(* Schneider Machine Expert - Basic project Prototype 2, file version 2.7.0.0 *)
(* ProjectInformations: Name=Nuevo proyecto *)

HARDWARE
  Cpu 0: TM221M16R/G
  EthernetConfiguration: NetworkName=M221, IpAllocationMode=FixedAddress, IpAddress=0.0.0.0, SubnetMask=0.0.0.0
  SerialLineConfiguration: Baud=Baud19200, Parity=ParityEven, DataBits=DataBits8, StopBits=StopBits1, PhysicalMedium=PhysicalMediumRs485, TransmissionMode=TransmissionModeModbusRtu, SlaveId=1, Addressing=SlaveAddressing
  MastTask: UsePeriodScanMode=false, PeriodScan=100
  FastTask: Period=255
  CpuBehavior: StartingMode=StartAsPreviousState, AutoSaveRamOnEeprom=true, WatchdogPeriod=250

SYMBOLS  (address, symbol, comment, settings)
  %M0       START_BUTTON
  %M1       RESET_BUTTON
  %M2       STOP_BUTTON
  %M3       EMERGENCY_BUTTON
  %M4       AUTO_SWITCH
  %M5       TYPE_2
  %M6       TYPE_3
  %M7       ENTRY_SENSOR
  %M8       OBJECT_SENSOR_1
  %M9       EXIT_SENSOR
  %M10      PERSON
  %M11      OBJECT_SENSOR_2
  %M12      T1_SENSOR
  %M13      T2_SENSOR
  %M14      T3_SENSOR
  %M15      ENTRY_CONVEYOR
  %M16      GRAB_1
  %M17      MIDDLE_CONVEYOR
  %M18      GRAB_2
  %M19      EXIT_CONVEYOR
  %M20      CURVE_CONVEYOR
  %M21      SELECTOR_CONVEYOR
  %M22      T1_CONVEYOR
  %M23      T2_CONVEYOR
  %M24      T3_CONVEYOR
  %M25      BELT_1
  %M26      BELT_2
  %M27      BELT_3
  %M28      PALLET
  %M29      RED
  %M30      YELLOW
  %M31      GREEN
  %M32      ALARM
  %M33      ENTRY
  %M100     INITIALIZE
  %M101     INITIAL_POS_1
  %M102     INITIAL_POS_2
  %M200     FLAG_AUTO
  %S21      SB_INITGRAFCET  "En el estado 1, este bit provoca una inicialización GRAFCET. Los pasos activos se desactivan y los pasos iniciales se activan"
  %X1       STATE_1
  %X2       STATE_2
  %X3       STATE_3
  %X4       STATE_4
  %X5       STATE_5
  %X6       STATE_6
  %X7       STATE_7
  %X8       STATE_8
  %X9       STATE_9
  %X10      STATE_10
  %X11      STATE_11
  %X12      STATE_12
  %X13      STATE_13
  %X14      STATE_14
  %X15      STATE_15
  %X16      STATE_16
  %X17      STATE_17
  %X18      STATE_18
  %X19      STATE_19
  %X21      STATE_21
  %MW0      X1
  %MW1      Y1
  %MW2      Z1
  %MW3      X2
  %MW4      Y2
  %MW5      Z2
  %MW6      X1_MOVE
  %MW7      Y1_MOVE
  %MW8      Z1_MOVE
  %MW9      X2_MOVE
  %MW10     Y2_MOVE
  %MW11     Z2_MOVE
  %MW12     T1
  %MW13     T2
  %MW14     T3
  %TM0      TIME_TO_UNGRAB  [Preset=1, Base=OneHundredMilliSeconds]
  %TM1      SECURITY_TIME  [Preset=5, Base=OneSecond]
  %TM2      TIME_TO_WAIT_NEXT  [Preset=2, Base=OneSecond]
  %C0       T1_ITEMS
  %C1       T2_ITEMS
  %C2       T3_ITEMS

GRAFCET Grafcet
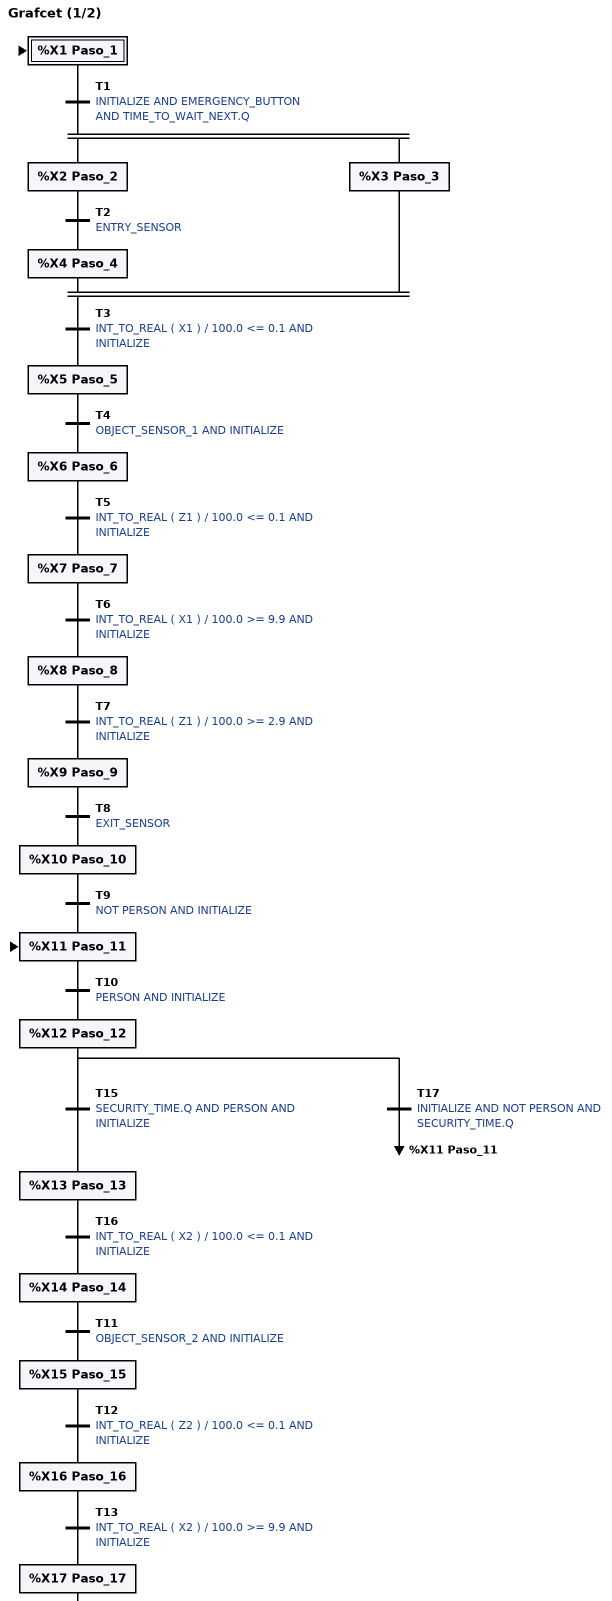
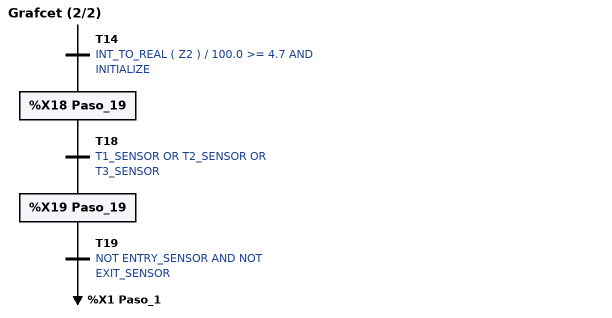
  INITIAL_STEP %X1  (* Paso_1 *)
  STEP %X2  (* Paso_2 *)
  STEP %X3  (* Paso_3 *)
  STEP %X4  (* Paso_4 *)
  STEP %X5  (* Paso_5 *)
  STEP %X6  (* Paso_6 *)
  STEP %X7  (* Paso_7 *)
  STEP %X8  (* Paso_8 *)
  STEP %X9  (* Paso_9 *)
  STEP %X10  (* Paso_10 *)
  STEP %X11  (* Paso_11 *)
  STEP %X12  (* Paso_12 *)
  STEP %X13  (* Paso_13 *)
  STEP %X14  (* Paso_14 *)
  STEP %X15  (* Paso_15 *)
  STEP %X16  (* Paso_16 *)
  STEP %X17  (* Paso_17 *)
  STEP %X18  (* Paso_19 *)
  STEP %X19  (* Paso_19 *)
  TRANSITION T1 FROM %X1 TO %X2, %X3 := INITIALIZE AND EMERGENCY_BUTTON AND TIME_TO_WAIT_NEXT.Q;
  TRANSITION T2 FROM %X2 TO %X4 := ENTRY_SENSOR;
  TRANSITION T3 FROM %X4, %X3 TO %X5 := INT_TO_REAL ( X1 ) / 100.0 <= 0.1 AND INITIALIZE;
  TRANSITION T4 FROM %X5 TO %X6 := OBJECT_SENSOR_1 AND INITIALIZE;
  TRANSITION T5 FROM %X6 TO %X7 := INT_TO_REAL ( Z1 ) / 100.0 <= 0.1 AND INITIALIZE;
  TRANSITION T6 FROM %X7 TO %X8 := INT_TO_REAL ( X1 ) / 100.0 >= 9.9 AND INITIALIZE;
  TRANSITION T7 FROM %X8 TO %X9 := INT_TO_REAL ( Z1 ) / 100.0 >= 2.9 AND INITIALIZE;
  TRANSITION T8 FROM %X9 TO %X10 := EXIT_SENSOR;
  TRANSITION T9 FROM %X10 TO %X11 := NOT PERSON AND INITIALIZE;
  TRANSITION T10 FROM %X11 TO %X12 := PERSON AND INITIALIZE;
  TRANSITION T11 FROM %X14 TO %X15 := OBJECT_SENSOR_2 AND INITIALIZE;
  TRANSITION T12 FROM %X15 TO %X16 := INT_TO_REAL ( Z2 ) / 100.0 <= 0.1 AND INITIALIZE;
  TRANSITION T13 FROM %X16 TO %X17 := INT_TO_REAL ( X2 ) / 100.0 >= 9.9 AND INITIALIZE;
  TRANSITION T14 FROM %X17 TO %X18 := INT_TO_REAL ( Z2 ) / 100.0 >= 4.7 AND INITIALIZE;
  TRANSITION T15 FROM %X12 TO %X13 := SECURITY_TIME.Q AND PERSON AND INITIALIZE;
  TRANSITION T16 FROM %X13 TO %X14 := INT_TO_REAL ( X2 ) / 100.0 <= 0.1 AND INITIALIZE;
  TRANSITION T17 FROM %X12 TO %X11 := INITIALIZE AND NOT PERSON AND SECURITY_TIME.Q;
  TRANSITION T18 FROM %X18 TO %X19 := T1_SENSOR OR T2_SENSOR OR T3_SENSOR;
  TRANSITION T19 FROM %X19 TO %X1 := NOT ENTRY_SENSOR AND NOT EXIT_SENSOR;

TRANSITION T1 (%X1 -> %X2, %X3) 
  (* SectionNumber=0 *)

// Rung 0: Tr1
  LD %M100                (* INITIALIZE *)
  AND %M3                 (* EMERGENCY_BUTTON *)
  AND %TM2.Q              (* TIME_TO_WAIT_NEXT *)
  ENDT
  // as ST:
  //   TRANSITION := INITIALIZE AND EMERGENCY_BUTTON AND TIME_TO_WAIT_NEXT.Q;

TRANSITION T2 (%X2 -> %X4) 
  (* SectionNumber=0 *)

// Rung 1: Tr2
  LD %M7                  (* ENTRY_SENSOR *)
  ENDT
  // as ST:
  //   TRANSITION := ENTRY_SENSOR;

TRANSITION T3 (%X4, %X3 -> %X5) 
  (* SectionNumber=0 *)

// Rung 2: Tr3
  LD 1
  AND [ INT_TO_REAL ( %MW0 ) / 100.0 <= 0.1 ](* X1 *)
  AND %M100               (* INITIALIZE *)
  ENDT
  // as ST:
  //   TRANSITION := INT_TO_REAL ( X1 ) / 100.0 <= 0.1 AND INITIALIZE;

TRANSITION T4 (%X5 -> %X6) 
  (* SectionNumber=0 *)

// Rung 3: Tr4
  LD %M8                  (* OBJECT_SENSOR_1 *)
  AND %M100               (* INITIALIZE *)
  ENDT
  // as ST:
  //   TRANSITION := OBJECT_SENSOR_1 AND INITIALIZE;

TRANSITION T5 (%X6 -> %X7) 
  (* SectionNumber=0 *)

// Rung 4: Tr5
  LD 1
  AND [ INT_TO_REAL ( %MW2 ) / 100.0 <= 0.1 ](* Z1 *)
  AND %M100               (* INITIALIZE *)
  ENDT
  // as ST:
  //   TRANSITION := INT_TO_REAL ( Z1 ) / 100.0 <= 0.1 AND INITIALIZE;

TRANSITION T6 (%X7 -> %X8) 
  (* SectionNumber=0 *)

// Rung 5: Tr6
  LD 1
  AND [ INT_TO_REAL ( %MW0 ) / 100.0 >= 9.9 ](* X1 *)
  AND %M100               (* INITIALIZE *)
  ENDT
  // as ST:
  //   TRANSITION := INT_TO_REAL ( X1 ) / 100.0 >= 9.9 AND INITIALIZE;

TRANSITION T7 (%X8 -> %X9) 
  (* SectionNumber=0 *)

// Rung 6: Tr7
  LD 1
  AND [ INT_TO_REAL ( %MW2 ) / 100.0 >= 2.9 ](* Z1 *)
  AND %M100               (* INITIALIZE *)
  ENDT
  // as ST:
  //   TRANSITION := INT_TO_REAL ( Z1 ) / 100.0 >= 2.9 AND INITIALIZE;

TRANSITION T8 (%X9 -> %X10) 
  (* SectionNumber=0 *)

// Rung 7: Tr8
  LD %M9                  (* EXIT_SENSOR *)
  ENDT
  // as ST:
  //   TRANSITION := EXIT_SENSOR;

TRANSITION T9 (%X10 -> %X11) 
  (* SectionNumber=0 *)

// Rung 8: Tr9
  LDN %M10                (* PERSON *)
  AND %M100               (* INITIALIZE *)
  ENDT
  // as ST:
  //   TRANSITION := NOT PERSON AND INITIALIZE;

TRANSITION T10 (%X11 -> %X12) 
  (* SectionNumber=0 *)

// Rung 9: Tr10
  LD %M10                 (* PERSON *)
  AND %M100               (* INITIALIZE *)
  ENDT
  // as ST:
  //   TRANSITION := PERSON AND INITIALIZE;

TRANSITION T11 (%X14 -> %X15) 
  (* SectionNumber=0 *)

// Rung 10: Tr14
  LD %M11                 (* OBJECT_SENSOR_2 *)
  AND %M100               (* INITIALIZE *)
  ENDT
  // as ST:
  //   TRANSITION := OBJECT_SENSOR_2 AND INITIALIZE;

TRANSITION T12 (%X15 -> %X16) 
  (* SectionNumber=0 *)

// Rung 11: Tr15
  LD 1
  AND [ INT_TO_REAL ( %MW5 ) / 100.0 <= 0.1 ](* Z2 *)
  AND %M100               (* INITIALIZE *)
  ENDT
  // as ST:
  //   TRANSITION := INT_TO_REAL ( Z2 ) / 100.0 <= 0.1 AND INITIALIZE;

TRANSITION T13 (%X16 -> %X17) 
  (* SectionNumber=0 *)

// Rung 12: Tr16
  LD 1
  AND [ INT_TO_REAL ( %MW3 ) / 100.0 >= 9.9 ](* X2 *)
  AND %M100               (* INITIALIZE *)
  ENDT
  // as ST:
  //   TRANSITION := INT_TO_REAL ( X2 ) / 100.0 >= 9.9 AND INITIALIZE;

TRANSITION T14 (%X17 -> %X18) 
  (* SectionNumber=0 *)

// Rung 13: Tr17
  LD 1
  AND [ INT_TO_REAL ( %MW5 ) / 100.0 >= 4.7 ](* Z2 *)
  AND %M100               (* INITIALIZE *)
  ENDT
  // as ST:
  //   TRANSITION := INT_TO_REAL ( Z2 ) / 100.0 >= 4.7 AND INITIALIZE;

TRANSITION T15 (%X12 -> %X13) 
  (* SectionNumber=0 *)

// Rung 14: Tr12
  LD %TM1.Q               (* SECURITY_TIME *)
  AND %M10                (* PERSON *)
  AND %M100               (* INITIALIZE *)
  ENDT
  // as ST:
  //   TRANSITION := SECURITY_TIME.Q AND PERSON AND INITIALIZE;

TRANSITION T16 (%X13 -> %X14) 
  (* SectionNumber=0 *)

// Rung 15: Tr13
  LD 1
  AND [ INT_TO_REAL ( %MW3 ) / 100.0 <= 0.1 ](* X2 *)
  AND %M100               (* INITIALIZE *)
  ENDT
  // as ST:
  //   TRANSITION := INT_TO_REAL ( X2 ) / 100.0 <= 0.1 AND INITIALIZE;

TRANSITION T17 (%X12 -> %X11) 
  (* SectionNumber=0 *)

// Rung 16: Tr11
  LD %M100                (* INITIALIZE *)
  ANDN %M10               (* PERSON *)
  AND %TM1.Q              (* SECURITY_TIME *)
  ENDT
  // as ST:
  //   TRANSITION := INITIALIZE AND NOT PERSON AND SECURITY_TIME.Q;

TRANSITION T18 (%X18 -> %X19) 
  (* SectionNumber=0 *)

// Rung 17: Tr18
  LD %M12                 (* T1_SENSOR *)
  OR %M13                 (* T2_SENSOR *)
  OR %M14                 (* T3_SENSOR *)
  ENDT
  // as ST:
  //   TRANSITION := T1_SENSOR OR T2_SENSOR OR T3_SENSOR;

TRANSITION T19 (%X19 -> %X1) 
  (* SectionNumber=0 *)

// Rung 18: Tr19
  LDN %M7                 (* ENTRY_SENSOR *)
  ANDN %M9                (* EXIT_SENSOR *)
  ENDT
  // as ST:
  //   TRANSITION := NOT ENTRY_SENSOR AND NOT EXIT_SENSOR;

POU Actions
  (* SectionNumber=21 *)

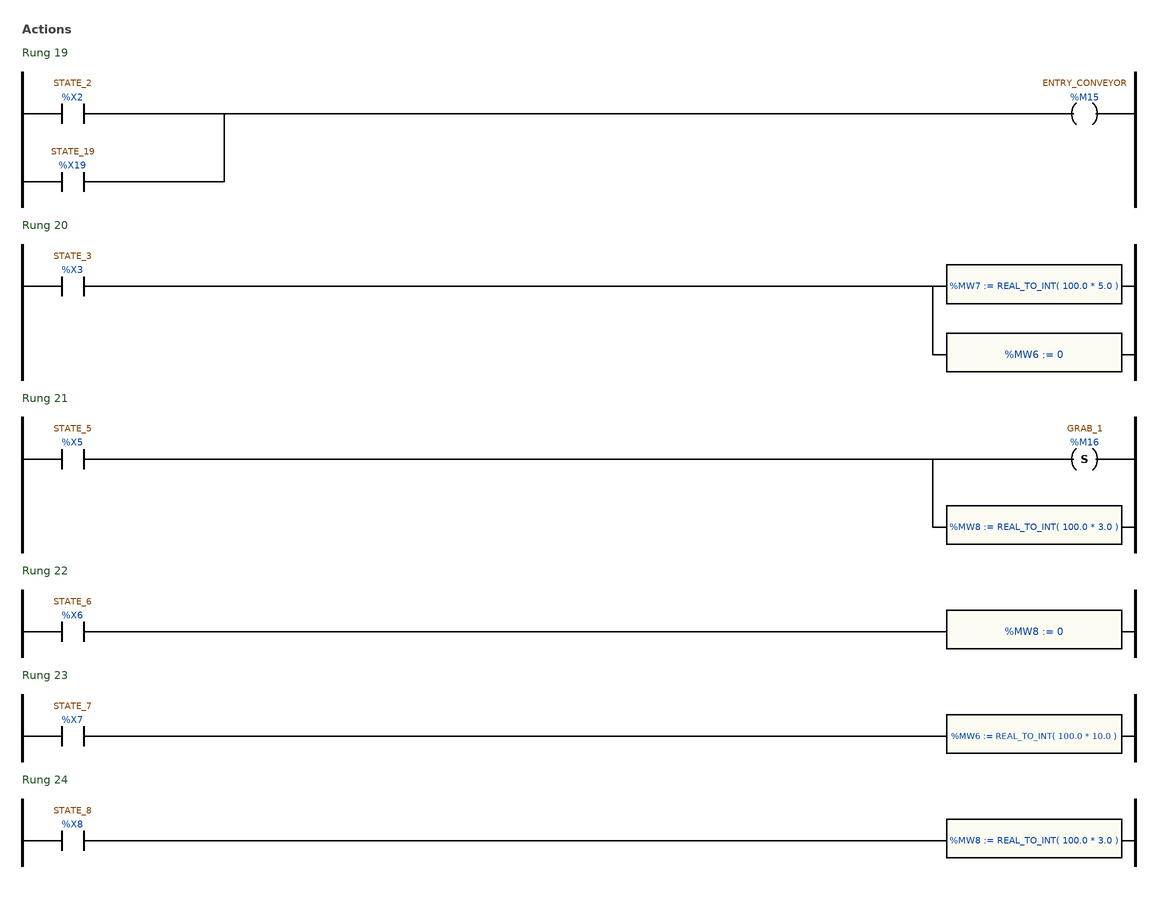

// Rung 19
  LD %X2                  (* STATE_2 *)
  OR %X19                 (* STATE_19 *)
  ST %M15                 (* ENTRY_CONVEYOR *)
  // as ST:
  //   ENTRY_CONVEYOR := STATE_2 OR STATE_19;

// Rung 20
  LD %X3                  (* STATE_3 *)
  [ %MW7 := REAL_TO_INT ( 100.0 * 5.0 ) ](* Y1_MOVE *)
  [ %MW6 := 0 ]           (* X1_MOVE *)
  // as ST:
  //   IF STATE_3 THEN Y1_MOVE := REAL_TO_INT ( 100.0 * 5.0 ); END_IF;
  //   IF STATE_3 THEN X1_MOVE := 0; END_IF;

// Rung 21
  LD %X5                  (* STATE_5 *)
  S %M16                  (* GRAB_1 *)
  [ %MW8 := REAL_TO_INT ( 100.0 * 3.0 ) ](* Z1_MOVE *)
  // as ST:
  //   IF STATE_5 THEN GRAB_1 := TRUE; END_IF;
  //   IF STATE_5 THEN Z1_MOVE := REAL_TO_INT ( 100.0 * 3.0 ); END_IF;

// Rung 22
  LD %X6                  (* STATE_6 *)
  [ %MW8 := 0 ]           (* Z1_MOVE *)
  // as ST:
  //   IF STATE_6 THEN Z1_MOVE := 0; END_IF;

// Rung 23
  LD %X7                  (* STATE_7 *)
  [ %MW6 := REAL_TO_INT ( 100.0 * 10.0 ) ](* X1_MOVE *)
  // as ST:
  //   IF STATE_7 THEN X1_MOVE := REAL_TO_INT ( 100.0 * 10.0 ); END_IF;

// Rung 24
  LD %X8                  (* STATE_8 *)
  [ %MW8 := REAL_TO_INT ( 100.0 * 3.0 ) ](* Z1_MOVE *)
  // as ST:
  //   IF STATE_8 THEN Z1_MOVE := REAL_TO_INT ( 100.0 * 3.0 ); END_IF;

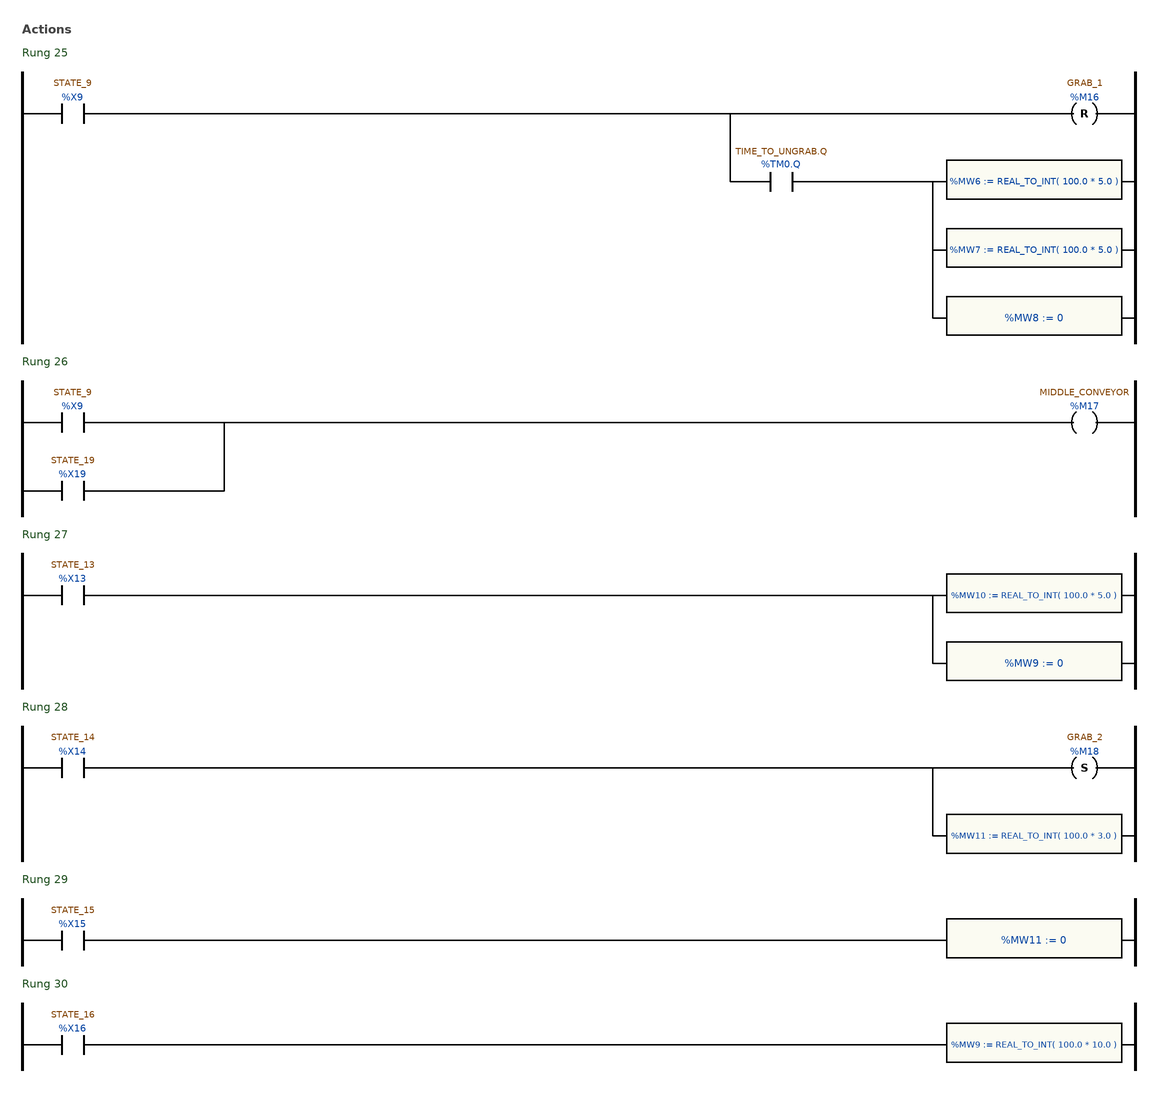

// Rung 25
  LD %X9                  (* STATE_9 *)
  MPS
  R %M16                  (* GRAB_1 *)
  MPP
  AND %TM0.Q              (* TIME_TO_UNGRAB *)
  [ %MW6 := REAL_TO_INT ( 100.0 * 5.0 ) ](* X1_MOVE *)
  [ %MW7 := REAL_TO_INT ( 100.0 * 5.0 ) ](* Y1_MOVE *)
  [ %MW8 := 0 ]           (* Z1_MOVE *)
  // as ST:
  //   IF STATE_9 THEN GRAB_1 := FALSE; END_IF;
  //   IF STATE_9 AND TIME_TO_UNGRAB.Q THEN X1_MOVE := REAL_TO_INT ( 100.0 * 5.0 ); END_IF;
  //   IF STATE_9 AND TIME_TO_UNGRAB.Q THEN Y1_MOVE := REAL_TO_INT ( 100.0 * 5.0 ); END_IF;
  //   IF STATE_9 AND TIME_TO_UNGRAB.Q THEN Z1_MOVE := 0; END_IF;

// Rung 26
  LD %X9                  (* STATE_9 *)
  OR %X19                 (* STATE_19 *)
  ST %M17                 (* MIDDLE_CONVEYOR *)
  // as ST:
  //   MIDDLE_CONVEYOR := STATE_9 OR STATE_19;

// Rung 27
  LD %X13                 (* STATE_13 *)
  [ %MW10 := REAL_TO_INT ( 100.0 * 5.0 ) ](* Y2_MOVE *)
  [ %MW9 := 0 ]           (* X2_MOVE *)
  // as ST:
  //   IF STATE_13 THEN Y2_MOVE := REAL_TO_INT ( 100.0 * 5.0 ); END_IF;
  //   IF STATE_13 THEN X2_MOVE := 0; END_IF;

// Rung 28
  LD %X14                 (* STATE_14 *)
  S %M18                  (* GRAB_2 *)
  [ %MW11 := REAL_TO_INT ( 100.0 * 3.0 ) ](* Z2_MOVE *)
  // as ST:
  //   IF STATE_14 THEN GRAB_2 := TRUE; END_IF;
  //   IF STATE_14 THEN Z2_MOVE := REAL_TO_INT ( 100.0 * 3.0 ); END_IF;

// Rung 29
  LD %X15                 (* STATE_15 *)
  [ %MW11 := 0 ]          (* Z2_MOVE *)
  // as ST:
  //   IF STATE_15 THEN Z2_MOVE := 0; END_IF;

// Rung 30
  LD %X16                 (* STATE_16 *)
  [ %MW9 := REAL_TO_INT ( 100.0 * 10.0 ) ](* X2_MOVE *)
  // as ST:
  //   IF STATE_16 THEN X2_MOVE := REAL_TO_INT ( 100.0 * 10.0 ); END_IF;

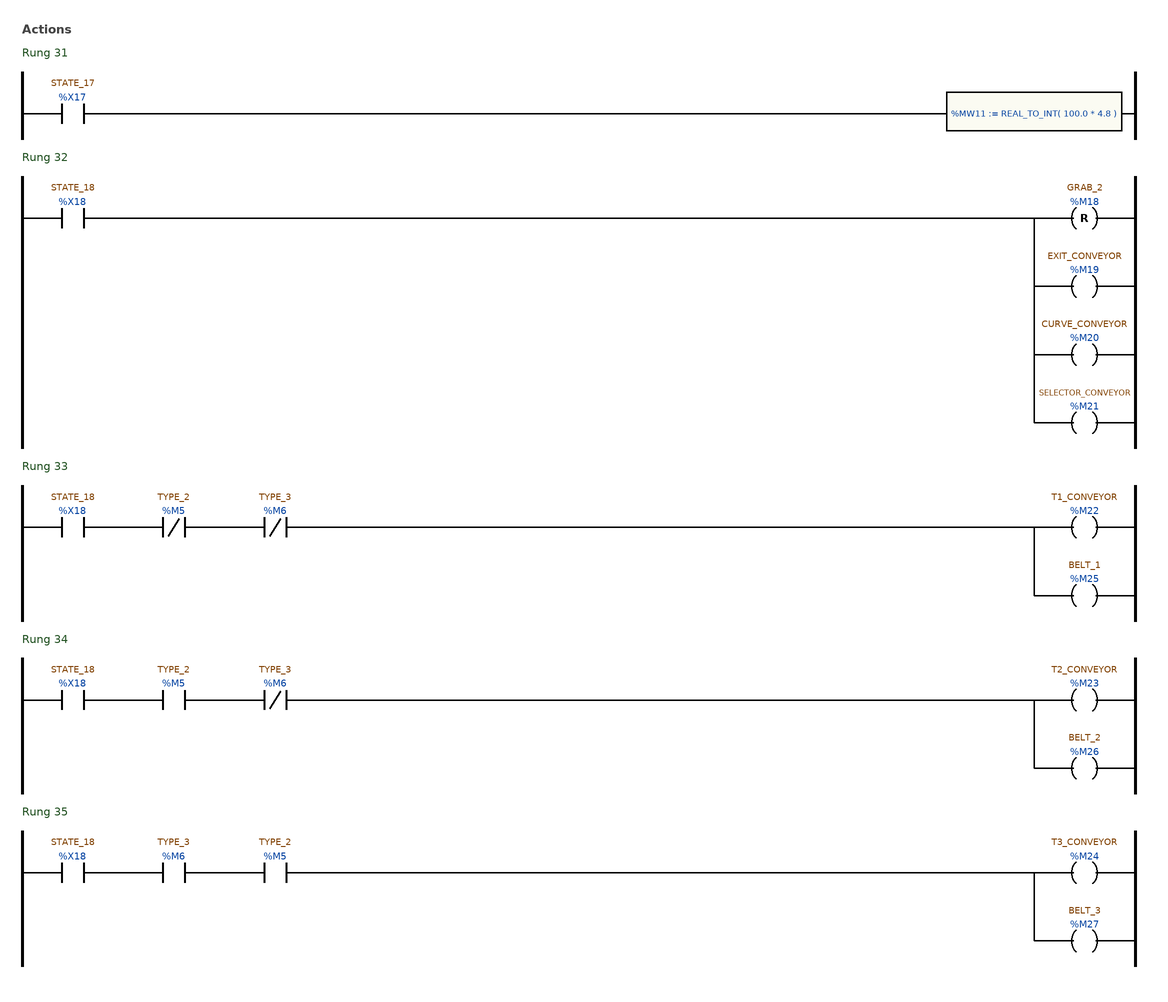

// Rung 31
  LD %X17                 (* STATE_17 *)
  [ %MW11 := REAL_TO_INT ( 100.0 * 4.8 ) ](* Z2_MOVE *)
  // as ST:
  //   IF STATE_17 THEN Z2_MOVE := REAL_TO_INT ( 100.0 * 4.8 ); END_IF;

// Rung 32
  LD %X18                 (* STATE_18 *)
  R %M18                  (* GRAB_2 *)
  ST %M19                 (* EXIT_CONVEYOR *)
  ST %M20                 (* CURVE_CONVEYOR *)
  ST %M21                 (* SELECTOR_CONVEYOR *)
  // as ST:
  //   IF STATE_18 THEN GRAB_2 := FALSE; END_IF;
  //   EXIT_CONVEYOR := STATE_18;
  //   CURVE_CONVEYOR := STATE_18;
  //   SELECTOR_CONVEYOR := STATE_18;

// Rung 33
  LD %X18                 (* STATE_18 *)
  ANDN %M5                (* TYPE_2 *)
  ANDN %M6                (* TYPE_3 *)
  ST %M22                 (* T1_CONVEYOR *)
  ST %M25                 (* BELT_1 *)
  // as ST:
  //   T1_CONVEYOR := STATE_18 AND NOT TYPE_2 AND NOT TYPE_3;
  //   BELT_1 := STATE_18 AND NOT TYPE_2 AND NOT TYPE_3;

// Rung 34
  LD %X18                 (* STATE_18 *)
  AND %M5                 (* TYPE_2 *)
  ANDN %M6                (* TYPE_3 *)
  ST %M23                 (* T2_CONVEYOR *)
  ST %M26                 (* BELT_2 *)
  // as ST:
  //   T2_CONVEYOR := STATE_18 AND TYPE_2 AND NOT TYPE_3;
  //   BELT_2 := STATE_18 AND TYPE_2 AND NOT TYPE_3;

// Rung 35
  LD %X18                 (* STATE_18 *)
  AND %M6                 (* TYPE_3 *)
  AND %M5                 (* TYPE_2 *)
  ST %M24                 (* T3_CONVEYOR *)
  ST %M27                 (* BELT_3 *)
  // as ST:
  //   T3_CONVEYOR := STATE_18 AND TYPE_3 AND TYPE_2;
  //   BELT_3 := STATE_18 AND TYPE_3 AND TYPE_2;

POU Buttons
  (* SectionNumber=22 *)

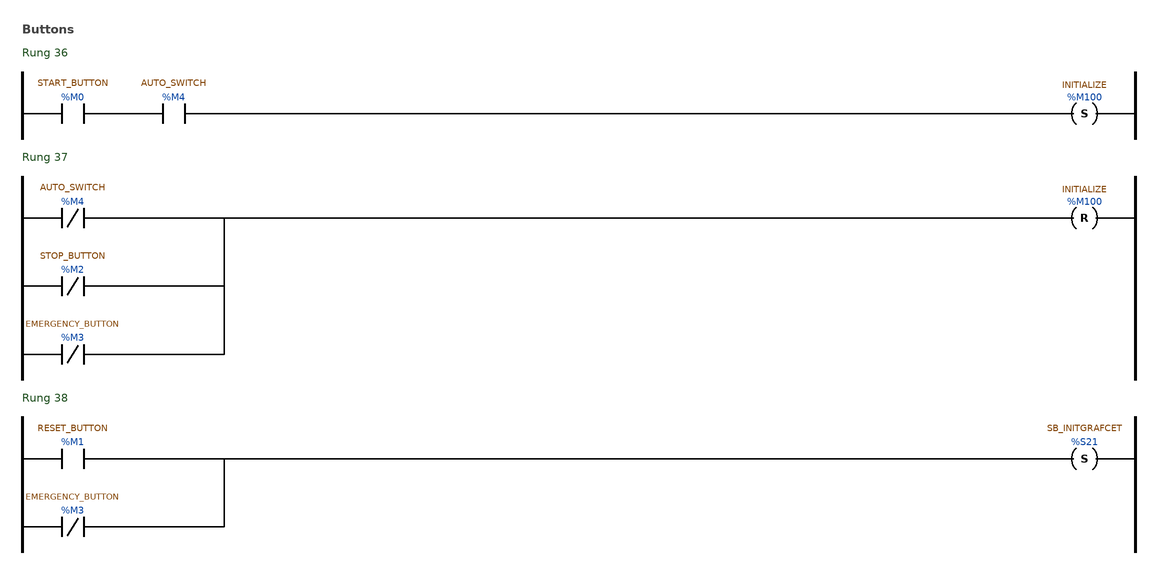

// Rung 36
  LD %M0                  (* START_BUTTON *)
  AND %M4                 (* AUTO_SWITCH *)
  S %M100                 (* INITIALIZE *)
  // as ST:
  //   IF START_BUTTON AND AUTO_SWITCH THEN INITIALIZE := TRUE; END_IF;

// Rung 37
  LDN %M4                 (* AUTO_SWITCH *)
  ORN %M2                 (* STOP_BUTTON *)
  ORN %M3                 (* EMERGENCY_BUTTON *)
  R %M100                 (* INITIALIZE *)
  // as ST:
  //   IF NOT AUTO_SWITCH OR NOT STOP_BUTTON OR NOT EMERGENCY_BUTTON THEN INITIALIZE := FALSE; END_IF;

// Rung 38
  LD %M1                  (* RESET_BUTTON *)
  ORN %M3                 (* EMERGENCY_BUTTON *)
  S %S21                  (* SB_INITGRAFCET *)
  // as ST:
  //   IF RESET_BUTTON OR NOT EMERGENCY_BUTTON THEN SB_INITGRAFCET := TRUE; END_IF;

POU Timers and Counters
  (* SectionNumber=23 *)

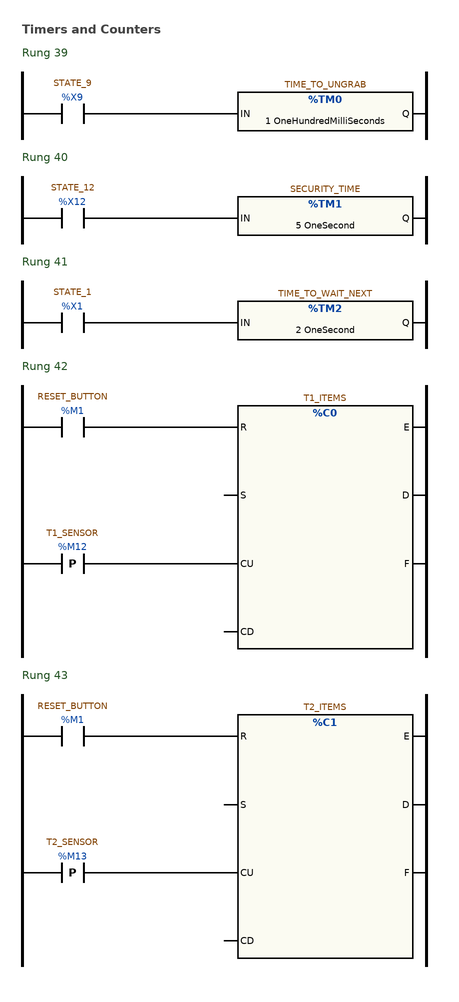

// Rung 39
  BLK %TM0                (* TIME_TO_UNGRAB *)
  LD %X9                  (* STATE_9 *)
  IN
  END_BLK
  // as ST:
  //   TIME_TO_UNGRAB(IN := STATE_9);

// Rung 40
  BLK %TM1                (* SECURITY_TIME *)
  LD %X12                 (* STATE_12 *)
  IN
  END_BLK
  // as ST:
  //   SECURITY_TIME(IN := STATE_12);

// Rung 41
  BLK %TM2                (* TIME_TO_WAIT_NEXT *)
  LD %X1                  (* STATE_1 *)
  IN
  END_BLK
  // as ST:
  //   TIME_TO_WAIT_NEXT(IN := STATE_1);

// Rung 42
  BLK %C0                 (* T1_ITEMS *)
  LD %M1                  (* RESET_BUTTON *)
  R
  LDR %M12                (* T1_SENSOR *)
  CU
  END_BLK
  // as ST:
  //   T1_ITEMS(R := RESET_BUTTON, CU := RISING(T1_SENSOR));

// Rung 43
  BLK %C1                 (* T2_ITEMS *)
  LD %M1                  (* RESET_BUTTON *)
  R
  LDR %M13                (* T2_SENSOR *)
  CU
  END_BLK
  // as ST:
  //   T2_ITEMS(R := RESET_BUTTON, CU := RISING(T2_SENSOR));

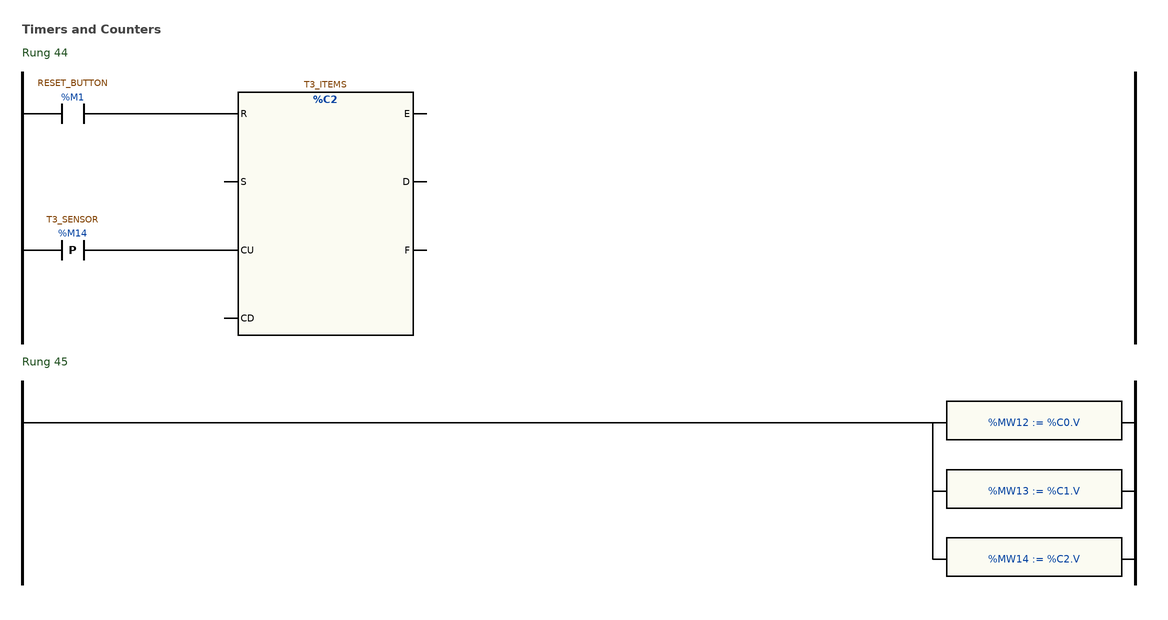

// Rung 44
  BLK %C2                 (* T3_ITEMS *)
  LD %M1                  (* RESET_BUTTON *)
  R
  LDR %M14                (* T3_SENSOR *)
  CU
  END_BLK
  // as ST:
  //   T3_ITEMS(R := RESET_BUTTON, CU := RISING(T3_SENSOR));

// Rung 45
  LD 1
  [ %MW12 := %C0.V ]      (* T1, T1_ITEMS *)
  [ %MW13 := %C1.V ]      (* T2, T2_ITEMS *)
  [ %MW14 := %C2.V ]      (* T3, T3_ITEMS *)
  // as ST:
  //   T1 := T1_ITEMS.V;
  //   T2 := T2_ITEMS.V;
  //   T3 := T3_ITEMS.V;

POU Initial conditions
  (* SectionNumber=24 *)

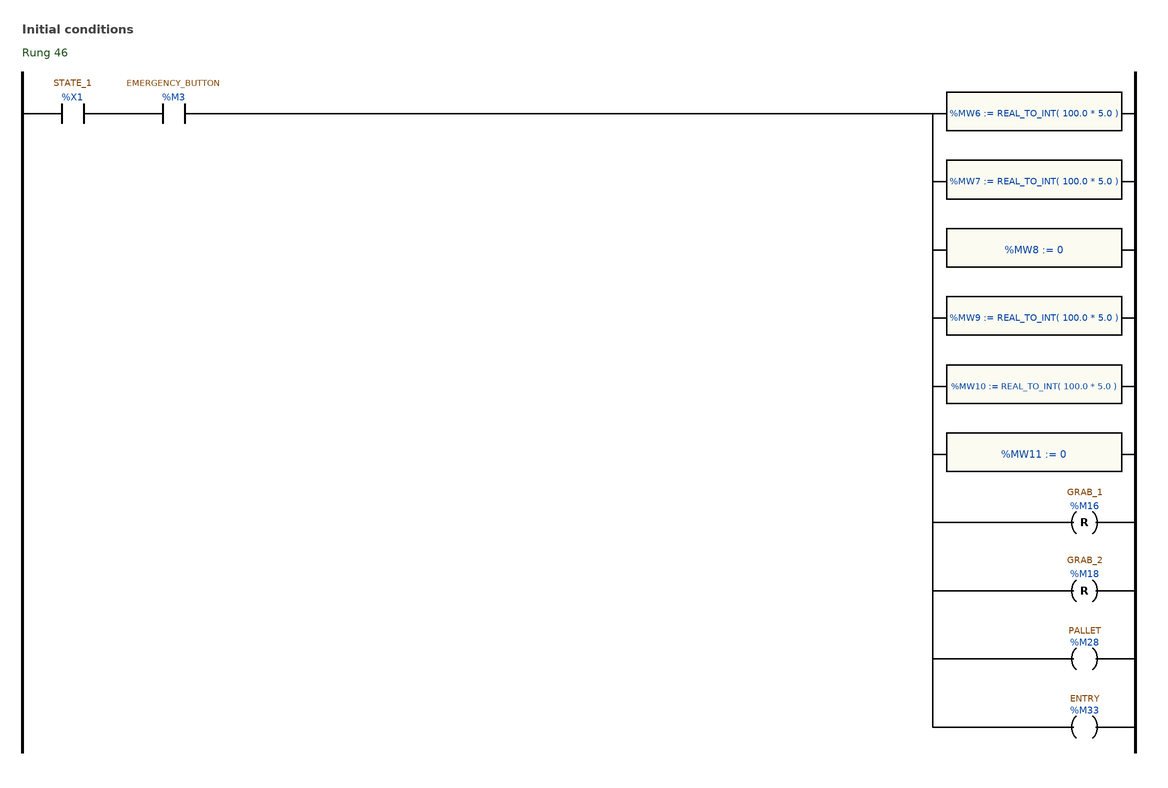

// Rung 46
  LD %X1                  (* STATE_1 *)
  AND %M3                 (* EMERGENCY_BUTTON *)
  [ %MW6 := REAL_TO_INT ( 100.0 * 5.0 ) ](* X1_MOVE *)
  [ %MW7 := REAL_TO_INT ( 100.0 * 5.0 ) ](* Y1_MOVE *)
  [ %MW8 := 0 ]           (* Z1_MOVE *)
  [ %MW9 := REAL_TO_INT ( 100.0 * 5.0 ) ](* X2_MOVE *)
  [ %MW10 := REAL_TO_INT ( 100.0 * 5.0 ) ](* Y2_MOVE *)
  [ %MW11 := 0 ]          (* Z2_MOVE *)
  R %M16                  (* GRAB_1 *)
  R %M18                  (* GRAB_2 *)
  ST %M28                 (* PALLET *)
  ST %M33                 (* ENTRY *)
  // as ST:
  //   IF STATE_1 AND EMERGENCY_BUTTON THEN X1_MOVE := REAL_TO_INT ( 100.0 * 5.0 ); END_IF;
  //   IF STATE_1 AND EMERGENCY_BUTTON THEN Y1_MOVE := REAL_TO_INT ( 100.0 * 5.0 ); END_IF;
  //   IF STATE_1 AND EMERGENCY_BUTTON THEN Z1_MOVE := 0; END_IF;
  //   IF STATE_1 AND EMERGENCY_BUTTON THEN X2_MOVE := REAL_TO_INT ( 100.0 * 5.0 ); END_IF;
  //   IF STATE_1 AND EMERGENCY_BUTTON THEN Y2_MOVE := REAL_TO_INT ( 100.0 * 5.0 ); END_IF;
  //   IF STATE_1 AND EMERGENCY_BUTTON THEN Z2_MOVE := 0; END_IF;
  //   IF STATE_1 AND EMERGENCY_BUTTON THEN GRAB_1 := FALSE; END_IF;
  //   IF STATE_1 AND EMERGENCY_BUTTON THEN GRAB_2 := FALSE; END_IF;
  //   PALLET := STATE_1 AND EMERGENCY_BUTTON;
  //   ENTRY := STATE_1 AND EMERGENCY_BUTTON;

POU Lights and warnings
  (* SectionNumber=25 *)

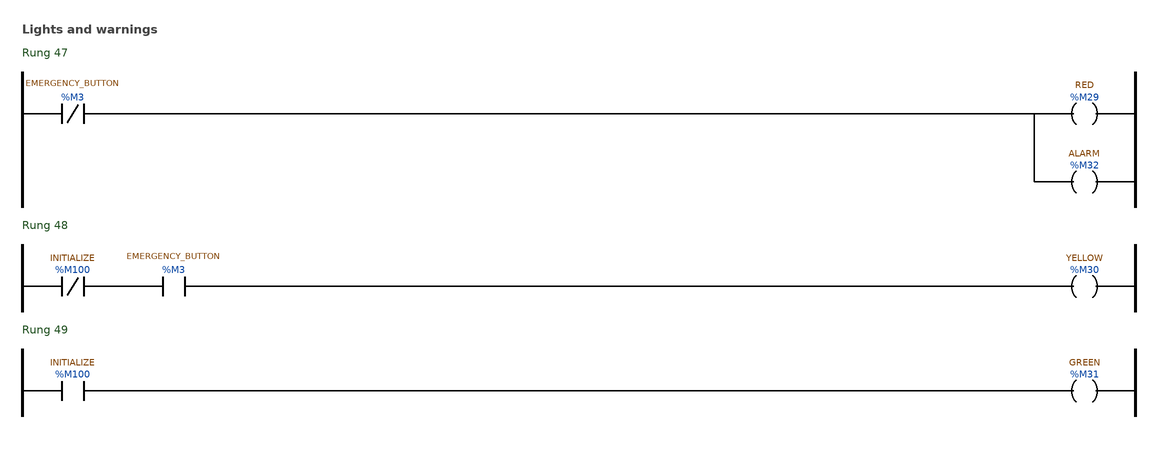

// Rung 47
  LDN %M3                 (* EMERGENCY_BUTTON *)
  ST %M29                 (* RED *)
  ST %M32                 (* ALARM *)
  // as ST:
  //   RED := NOT EMERGENCY_BUTTON;
  //   ALARM := NOT EMERGENCY_BUTTON;

// Rung 48
  LDN %M100               (* INITIALIZE *)
  AND %M3                 (* EMERGENCY_BUTTON *)
  ST %M30                 (* YELLOW *)
  // as ST:
  //   YELLOW := NOT INITIALIZE AND EMERGENCY_BUTTON;

// Rung 49
  LD %M100                (* INITIALIZE *)
  ST %M31                 (* GREEN *)
  // as ST:
  //   GREEN := INITIALIZE;
